(* PLC project Tc2_Utilities.BE32_TO_HOST Demo, tc3-libraries-kb TwinCAT 3.1 *)
(* stored: creationDateTime 2026-05-10T11:00:00, modificationDateTime 2026-05-10T11:00:00 *)

PROGRAM P_Demo_BE32_TO_HOST
  VAR
    bResult : DWORD;  (* BE32_TO_HOST 的返回值 *)
    bRun : BOOL;  (* 触发一次调用 *)
  END_VAR

            // ============================================================
// Tc2_Utilities.BE32_TO_HOST 演示程序（FUNCTION）
// ============================================================
// 验证步骤：
//   1. 引用 Tc2_Utilities（及依赖类型所在的库）
//   2. 编译 + 登录
//   3. 强制 bRun := TRUE 一个周期
//   4. 观察 bResult 应为 16#12345678
// ============================================================

IF bRun THEN
    bResult := BE32_TO_HOST(16#78563412);
    bRun := FALSE;
END_IF;

          
END_PROGRAM
